FUNCTION_BLOCK T_CantChangeModInExecute EXTENDS T_UnitTestBase
VAR
  em : EquipmentModule;
  actual, expected : E_PMLUnitMode;
  actualState, expectedState : E_PMLState;
  scanCounter : INT;
  myTestState : (ARRANGE, ACT, ASSERT);
END_VAR

CASE myTestState OF

  ARRANGE:
    em.CyclicLogic();

    IF em.InitComplete THEN
      myTestState := ACT;
      em.ChangeState(E_PMLCommand.ePMLCommand_Clear);
    END_IF

    CycleModuleLogicToAllowChangesToFilterThrough();
    em.ChangeState(E_PMLCommand.ePMLCommand_Reset);

    CycleModuleLogicToAllowChangesToFilterThrough();
    em.ChangeState(E_PMLCommand.ePMLCommand_Start);
    CycleModuleLogicToAllowChangesToFilterThrough();

  ACT:
      
    em.ChangeMode(E_PMLUnitMode.ePMLUnitMode_Maintenance);
    CycleModuleLogicToAllowChangesToFilterThrough();

    actual := em.CurrentMode;
    expected := E_PMLUnitMode.ePMLUnitMode_Production;
    myTestState := ASSERT;
    
    actualState := em.CurrentState;
    expectedState := E_PMLState.ePMLState_Execute;

  ASSERT:
    assertion.AssertEquals_UINT(TO_UINT(expected), TO_UINT(actual), 'actualState := em.CurrentState;');
    assertion.AssertEquals_UINT(TO_UINT(actual), TO_UINT(expected), 'actual := em.CurrentMode');
    myTestState := ARRANGE;
    TestFinished();

END_CASE

METHOD CycleModuleLogicToAllowChangesToFilterThrough : BOOL
VAR_INST
	i: INT;

END_VAR
//em.CyclicLogic();
//CycleModuleLogicToAllowChangesToFilterThrough := i >= 100;
//i := SEL(i >= 100, i + 1, 0);

FOR i := 0 TO 100 DO
  em.CyclicLogic();
END_FOR
END_METHOD

END_FUNCTION_BLOCK

(* stored: Version 1.1.0.1, ProductVersion 3.1.4024.12
   POU T_CantChangeModInExecute: Id {e2f5c05e-ff60-40d7-8f8a-a86764941221}, SpecialFunc None
   Method CycleModuleLogicToAllowChangesToFilterThrough: Id {a08e4b00-2491-4ffa-8bb6-7dc1f43a76c0} *)
